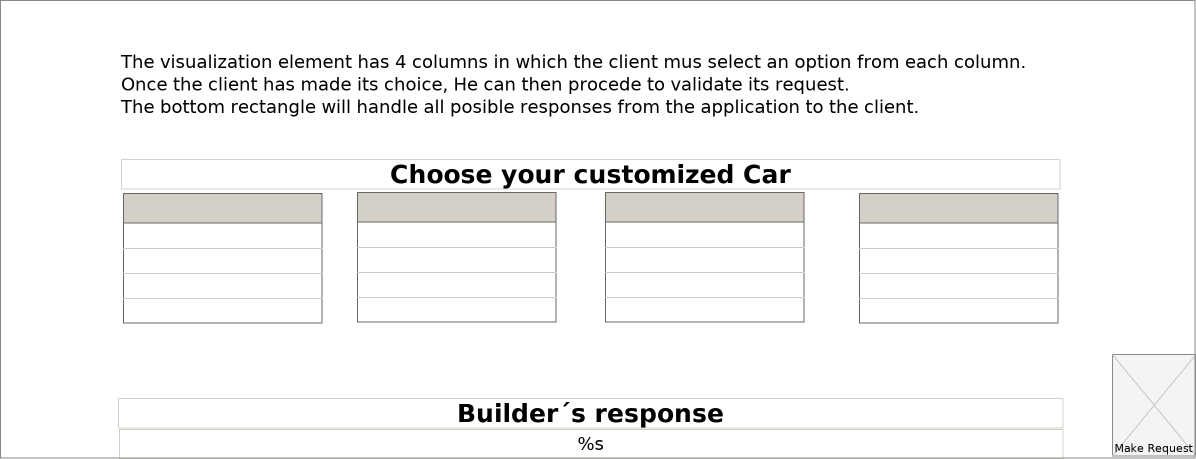
VISUALIZATION Visualization  // 1196x459
    Label (118,35 953x99), "The visualization element has 4 columns in which the client mus select an option from each column. Once the client has made its choice, He can then procede to validate its request. The bottom rectangle will handle all posible responses from the application to the client."
    Label (291,404 475x30)
    Image (1112,354 84x102), "Make Request", image: VisuSymbols.Symbols.OK
        OnMouseClick: toggle MAIN.bRequest
    Textfield (119,429 944x30), "%s", text variable: MAIN.sMessageLog
    Textfield (118,398 945x30), "Builder´s response"
    Textfield (121,159 939x30), "Choose your customized Car"
    Table (123,193 199x130), data array: MAIN.arrayChassis
        p3854506369: MAIN.arrayChassis[INDEX]
        p1892666644: MAIN.tableArray[2,INDEX]
        p338671338: MAIN.tableArray[3,INDEX]
        p2170511999: MAIN.tableArray[4,INDEX]
        p2232123230: Chassis Colour
        p511219082: Car type
        p1755163831: Motor dimensions
        p4092479075: Wheels type
        p1137915858: MAIN.iChassis
        p1822360349: MAIN.bChassis
    Table (357,192 199x130), data array: MAIN.arrayCarType
        p3854506369: MAIN.arrayCarType[INDEX]
        p1892666644: MAIN.tableArray[2,INDEX]
        p338671338: MAIN.tableArray[3,INDEX]
        p2170511999: MAIN.tableArray[4,INDEX]
        p2232123230: Car Type
        p511219082: Car type
        p1755163831: Motor dimensions
        p4092479075: Wheels type
        p1137915858: MAIN.iCarType
        p1822360349: MAIN.bCarType
    Table (605,192 199x130), data array: MAIN.arrayMotor
        p3854506369: MAIN.arrayMotor[INDEX]
        p1892666644: MAIN.tableArray[2,INDEX]
        p338671338: MAIN.tableArray[3,INDEX]
        p2170511999: MAIN.tableArray[4,INDEX]
        p2232123230: Motor Dimensions
        p511219082: Car type
        p1755163831: Motor dimensions
        p4092479075: Wheels type
        p1137915858: MAIN.iMotor
        p1822360349: MAIN.bMotor
    Table (859,193 199x130), data array: MAIN.arrayTires
        p3854506369: MAIN.arrayTires[INDEX]
        p1892666644: MAIN.tableArray[2,INDEX]
        p338671338: MAIN.tableArray[3,INDEX]
        p2170511999: MAIN.tableArray[4,INDEX]
        p511219082: Car type
        p1755163831: Motor dimensions
        p4092479075: Wheels type
        p1137915858: MAIN.iTires
        p1822360349: MAIN.bTires
END_VISUALIZATION

(* stored: Version 1.1.0.1, ProductVersion 3.1.4024.12
   Visu Visualization: Id {f537bab1-5750-421d-af35-343b31f2a5fe} *)
